PROGRAM main
VAR
	//attuatori
	AttuatBraccioGiu : BOOL := FALSE;
	AttuatBraccioSu : BOOL := FALSE;
	AttuatBraccioSx : BOOL := FALSE;
	AttuatBraccioDx : BOOL := FALSE;
	AttuatBraccioPresa : BOOL := FALSE;
	AttuatBraccioRilascio : BOOL := FALSE;
	AttuatRiempiSerbatoio : BOOL := FALSE;
	AttuatSvuotaSerbatoio : BOOL := FALSE;
	AttuatFinestra : BOOL := FALSE;
	AttuatCondizionatore : BOOL := FALSE;
	AttuatRullo : BOOL := FALSE;
	AttuatLampada : BOOL := FALSE;
	//sensori
	SensoreFCB : BOOL := FALSE;
	SensoreFCT : BOOL := FALSE;
	SensoreFCS : BOOL := FALSE;
	SensoreFCD : BOOL := FALSE;
	SensoreFineCorsaPianta2 : BOOL := FALSE;
	SensoreGrasp : BOOL := FALSE;
	SensoreRelease : BOOL := FALSE;
	SensoreRulloOccupato : BOOL := FALSE;
	SensoreVascaPienaVuota : BOOL := FALSE;
	SensoreSerbatoioOn : BOOL := FALSE;
	SensoreSerbatoioFull : BOOL := FALSE;
	SensoreSerbatoioEmpty : BOOL := FALSE;
	SensoreCondizionatore : BOOL := FALSE;
	SensoreLuci : BOOL := FALSE;
	SensoreFinestra : BOOL := FALSE;
	SensoreTempCalda : BOOL := FALSE;
	SensoreTempFredda : BOOL := FALSE;
	SensorePianta1Pronta : BOOL := FALSE;
	SensorePianta2Pronta : BOOL := FALSE;
	SensoreStart : BOOL := FALSE;
	SensoreReset : BOOL := FALSE;
	TemperaturaAttuale : INT;
	TemperaturaOttimale : INT := 36;
	durataGiorno : INT;
	durataNotte : INT;
	
	
	SerbatoioVuoto: BOOL;
	Pianta1Pronta: INT;
	TOK2: BOOL;
	SerbatoioPieno: BOOL;
	VascaVuota: BOOL;
	VascaPiena: BOOL;
	Pianta2Pronta: BOOL;
	RulloPieno: BOOL;
	SopraPianta1: INT;
	PrendiPianta1: BOOL;
	PosizionePianta1: BOOL;
	Pianta1Grasped: BOOL;
	Pianta1Sopra: BOOL;
	Pianta1Alzata: BOOL;
	Pianta1SopraRullo: BOOL;
	Pianta1SulRullo: INT;
	SulRullo: INT;
	Pianta1SulRulloSulRullo: BOOL;
	Pianta1Rilasciata: BOOL;
	SopraPianta2: INT;
END_VAR

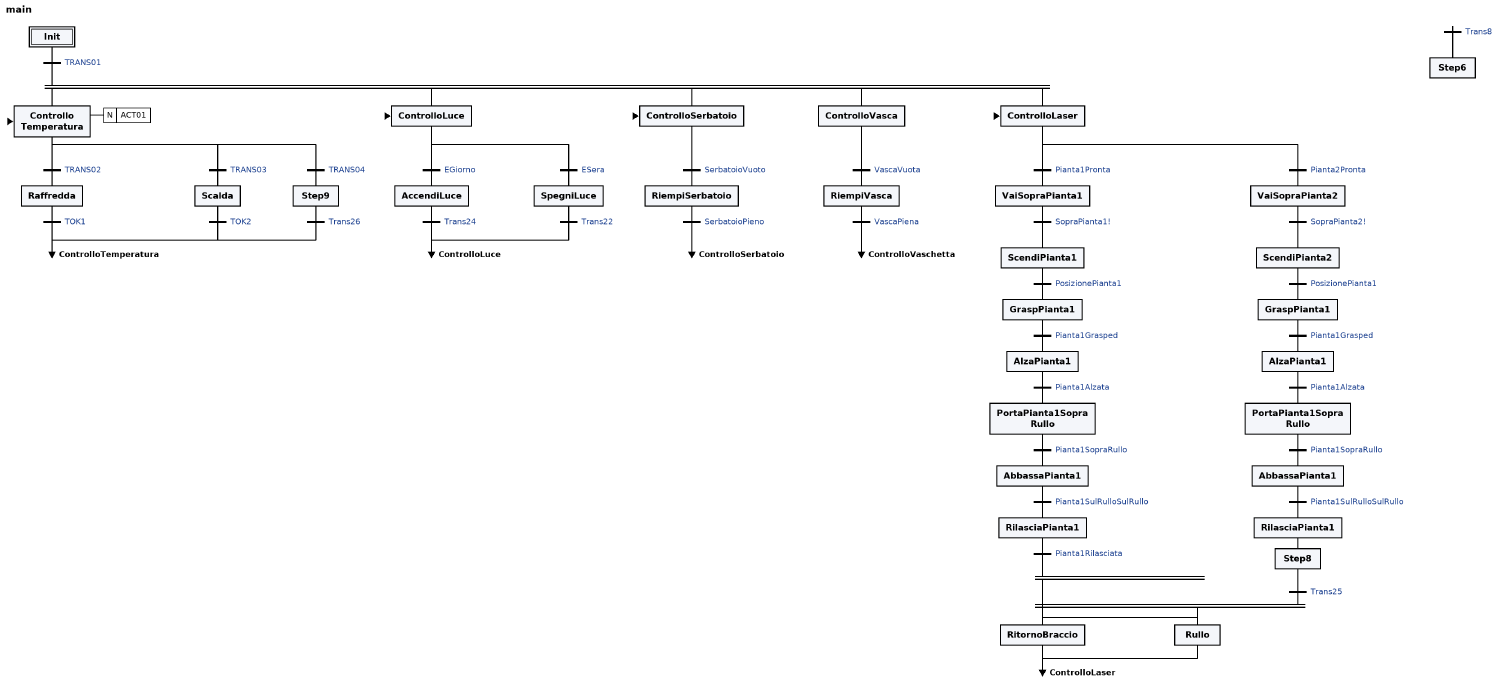
INITIAL_STEP Init:
END_STEP
TRANSITION FROM Init TO (ControlloTemperatura, ControlloLuce, ControlloSerbatoio, ControlloVasca, ControlloLaser)
    := TRANS01;
END_TRANSITION
STEP ControlloTemperatura:
    ACT01(N);
END_STEP
TRANSITION FROM ControlloTemperatura TO Raffredda
    := TRANS02;
END_TRANSITION
STEP Raffredda:
END_STEP
TRANSITION FROM Raffredda TO ControlloTemperatura
    := TOK1;
END_TRANSITION
TRANSITION FROM ControlloTemperatura TO Scalda
    := TRANS03;
END_TRANSITION
STEP Scalda:
END_STEP
TRANSITION FROM Scalda TO ControlloTemperatura
    := TOK2;
END_TRANSITION
TRANSITION FROM ControlloTemperatura TO Step9
    := TRANS04;
END_TRANSITION
STEP Step9:
END_STEP
TRANSITION FROM Step9 TO ControlloTemperatura
    := Trans26;
END_TRANSITION
STEP ControlloLuce:
END_STEP
TRANSITION FROM ControlloLuce TO AccendiLuce
    := EGiorno;
END_TRANSITION
STEP AccendiLuce:
END_STEP
TRANSITION FROM AccendiLuce TO ControlloLuce
    := Trans24;
END_TRANSITION
TRANSITION FROM ControlloLuce TO SpegniLuce
    := ESera;
END_TRANSITION
STEP SpegniLuce:
END_STEP
TRANSITION FROM SpegniLuce TO ControlloLuce
    := Trans22;
END_TRANSITION
STEP ControlloSerbatoio:
END_STEP
TRANSITION FROM ControlloSerbatoio TO RiempiSerbatoio
    := SerbatoioVuoto;
END_TRANSITION
STEP RiempiSerbatoio:
END_STEP
TRANSITION FROM RiempiSerbatoio TO ControlloSerbatoio
    := SerbatoioPieno;
END_TRANSITION
STEP ControlloVasca:
END_STEP
TRANSITION FROM ControlloVasca TO RiempiVasca
    := VascaVuota;
END_TRANSITION
STEP RiempiVasca:
END_STEP
TRANSITION FROM RiempiVasca TO ControlloVaschetta
    := VascaPiena;
END_TRANSITION
STEP ControlloLaser:
END_STEP
TRANSITION FROM ControlloLaser TO VaiSopraPianta1
    := Pianta1Pronta;
END_TRANSITION
STEP VaiSopraPianta1:
END_STEP
TRANSITION FROM VaiSopraPianta1 TO ScendiPianta1
    := SopraPianta1!;
END_TRANSITION
STEP ScendiPianta1:
END_STEP
TRANSITION FROM ScendiPianta1 TO GraspPianta1
    := PosizionePianta1;
END_TRANSITION
STEP GraspPianta1:
END_STEP
TRANSITION FROM GraspPianta1 TO AlzaPianta1
    := Pianta1Grasped;
END_TRANSITION
STEP AlzaPianta1:
END_STEP
TRANSITION FROM AlzaPianta1 TO PortaPianta1SopraRullo
    := Pianta1Alzata;
END_TRANSITION
STEP PortaPianta1SopraRullo:
END_STEP
TRANSITION FROM PortaPianta1SopraRullo TO AbbassaPianta1
    := Pianta1SopraRullo;
END_TRANSITION
STEP AbbassaPianta1:
END_STEP
TRANSITION FROM AbbassaPianta1 TO RilasciaPianta1
    := Pianta1SulRulloSulRullo;
END_TRANSITION
STEP RilasciaPianta1:
END_STEP
TRANSITION FROM RilasciaPianta1 TO (RitornoBraccio, Rullo)
    := Pianta1Rilasciata;
END_TRANSITION
TRANSITION FROM ControlloLaser TO VaiSopraPianta2
    := Pianta2Pronta;
END_TRANSITION
STEP VaiSopraPianta2:
END_STEP
TRANSITION FROM VaiSopraPianta2 TO ScendiPianta2
    := SopraPianta2!;
END_TRANSITION
STEP ScendiPianta2:
END_STEP
TRANSITION FROM ScendiPianta2 TO GraspPianta1
    := PosizionePianta1;
END_TRANSITION
STEP GraspPianta1:
END_STEP
TRANSITION FROM GraspPianta1 TO AlzaPianta1
    := Pianta1Grasped;
END_TRANSITION
STEP AlzaPianta1:
END_STEP
TRANSITION FROM AlzaPianta1 TO PortaPianta1SopraRullo
    := Pianta1Alzata;
END_TRANSITION
STEP PortaPianta1SopraRullo:
END_STEP
TRANSITION FROM PortaPianta1SopraRullo TO AbbassaPianta1
    := Pianta1SopraRullo;
END_TRANSITION
STEP AbbassaPianta1:
END_STEP
TRANSITION FROM AbbassaPianta1 TO RilasciaPianta1
    := Pianta1SulRulloSulRullo;
END_TRANSITION
STEP RilasciaPianta1:
END_STEP
// no transition between RilasciaPianta1 and Step8
STEP Step8:
END_STEP
TRANSITION FROM Step8 TO (RitornoBraccio, Rullo)
    := Trans25;
END_TRANSITION
STEP RitornoBraccio:
END_STEP
// no transition between RitornoBraccio and ControlloLaser
STEP Rullo:
END_STEP
// no transition between Rullo and ControlloLaser
TRANSITION FROM ??? TO Step6
    := Trans8;
END_TRANSITION
STEP Step6:
END_STEP

ACTION ACT01:
IF TemperaturaAttuale < TemperaturaOttimale-5 THEN
	SensoreTempFredda := TRUE;
	SensoreTempCalda := FALSE;
	
ELSIF TemperaturaAttuale > TemperaturaOttimale+5 THEN
	SensoreTempCalda := TRUE;
	SensoreTempFredda := FALSE;
END_IF
END_ACTION

TRANSITION TRANS01:
SensoreStart = TRUE AND SensoreFCTop= TRUE AND SensoreFCD = TRUE AND SensoreRulloOccupato = FALSE;
END_TRANSITION

TRANSITION TRANS02:
SensoreTempCalda := TRUE;
END_TRANSITION

TRANSITION TRANS03:
SensoreTempFredda := TRUE;
END_TRANSITION

TRANSITION TRANS04:
TemperaturaAttuale = TemperaturaOttimale;
END_TRANSITION

END_PROGRAM

(* stored: Version 1.1.0.1, ProductVersion 3.1.4024.15
   POU main: Id {b7796c3c-63d4-40cc-8177-a4d52dd478d6}, SpecialFunc None
   Action ACT01: Id {34dc420b-8947-4eec-a99d-0800aaf6b17a}
   Transition TRANS01: Id {58dfda41-c2f0-40b5-97e0-a48c1eae994f}
   Transition TRANS02: Id {fa3cf8e0-8591-4adf-b11d-d748c3d06fc1}
   Transition TRANS03: Id {b6f3ed56-5c9a-4f33-b947-956276a472c1}
   Transition TRANS04: Id {94dadf6a-ce5d-498f-980d-b2643ed6d930} *)
